{attribute 'GeneratedUsingTerminal: EL3356-0030-0025'}
{attribute addProperty BoxType "EL3356-0030-0025"}
{attribute addProperty Id "CtrlAT %Q*Ctrl_B9DDD3FF5"}
{attribute addProperty CRC "3427370076"}
{attribute addProperty Size "5"}
TYPE RMB_Control_CC49845C EXTENDS OutputBase_10CEE7DE :
STRUCT
	{attribute addProperty Name "Ctrl"}
	Ctrl AT %Q* : Ctrl_B9DDD3FF;
END_STRUCT
END_TYPE

(* stored: Version 1.2.0.0, ProductVersion 3.1.4024.11
   DUT RMB_Control_CC49845C: Id {2e08bc87-8db0-4675-acdb-7f7c941e4ad0} *)
